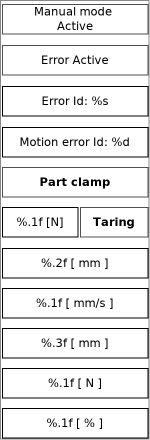
VISUALIZATION vHP3_AxisManualMode  // 150x440
VAR_IN_OUT
	fbData	: fbHP_Axis;
END_VAR
    Rectangle (2,207 76x30), "%.1f [N]", text variable: fbData.fbForceFilter.rOut
    Rectangle (2,4 146x30), "Manual mode Active", colour toggle: fbData.iWorkStep_Axis=15
    Rectangle (80,207 68x30), "Taring", colour toggle: fbData.bTaring, input disabled if: fbData.iWorkStep_Axis <> 15
        toggle fbData.bTaring p2164770859=TRUE
    Rectangle (2,45 146x30), "Error Active", colour toggle: fbData.IsErrorActive
    Rectangle (2,248 146x30), "%.2f [ mm ]", text variable: fbData.McReadActualPosition.Position
    Rectangle (2,167 146x30), "Part clamp", colour toggle: fbData.stInOuts.bQ_PartLockPiston, input disabled if: fbData.iWorkStep_Axis <> 15
        toggle fbData.stInOuts.bQ_PartLockPiston p2164770859=TRUE
    Rectangle (2,288 146x30), "%.1f [ mm/s ]", text variable: fbData.McReadActualVelocity.ActualVelocity
    Rectangle (2,86 146x30), "Error Id: %s", text variable: TO_STRING(fbData.nActEvent)
    Rectangle (2,127 146x30), "Motion error Id: %d", text variable: fbData.udiActErrorCode
    Rectangle (2,368 146x30), "%.1f [ N ]", text variable: fbData.stSettings.rManualModeMaxForceAtSlow
        OnMouseClick: write the text variable via Default, min 0, max 300, title 'Max force at slow manual move'
    Rectangle (2,408 146x30), "%.1f [ % ]", text variable: fbData.McTorqueMonitor.rTorqueLimit
        OnMouseClick: write the text variable via Default, min 1, max 100, title 'Motor torque limitation'
    Rectangle (2,328 146x30), "%.3f [ mm ]", text variable: fbData.lrCalibrationPoint_mm
END_VISUALIZATION

(* stored: Version 1.1.0.1, ProductVersion 3.1.4024.12
   Visu vHP3_AxisManualMode: Id {a47fbe6c-343f-4f28-8d7c-d2fc9153fb43} *)
